// SIMATIC S7-200 project (STEP 7-Micro/WIN), CPU 226 CN REL 02.01

ORGANIZATION_BLOCK 主程序:OB1
TITLE=程序注释
BEGIN
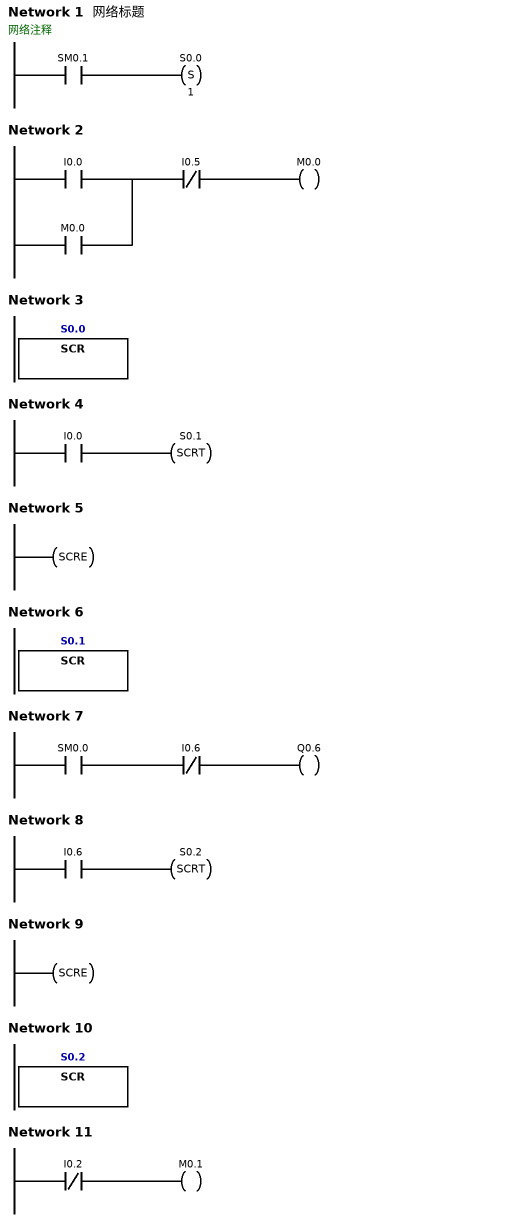
Network 1 // 网络标题
// 网络注释
LD     SM0.1
S      S0.0, 1
Network 2
LD     I0.0
O      M0.0
AN     I0.5
=      M0.0
Network 3
LSCR   S0.0
Network 4
LD     I0.0
SCRT   S0.1
Network 5
SCRE
Network 6
LSCR   S0.1
Network 7
LD     SM0.0
AN     I0.6
=      Q0.6
Network 8
LD     I0.6
SCRT   S0.2
Network 9
SCRE
Network 10
LSCR   S0.2
Network 11
LDN    I0.2
=      M0.1
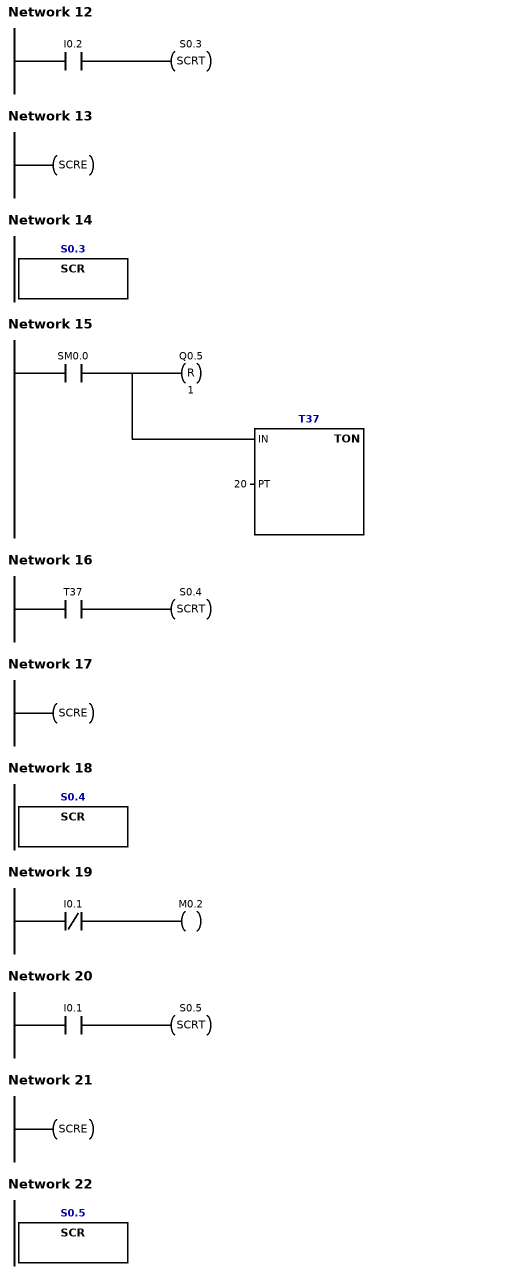
Network 12
LD     I0.2
SCRT   S0.3
Network 13
SCRE
Network 14
LSCR   S0.3
Network 15
LD     SM0.0
R      Q0.5, 1
TON    T37, 20
Network 16
LD     T37
SCRT   S0.4
Network 17
SCRE
Network 18
LSCR   S0.4
Network 19
LDN    I0.1
=      M0.2
Network 20
LD     I0.1
SCRT   S0.5
Network 21
SCRE
Network 22
LSCR   S0.5
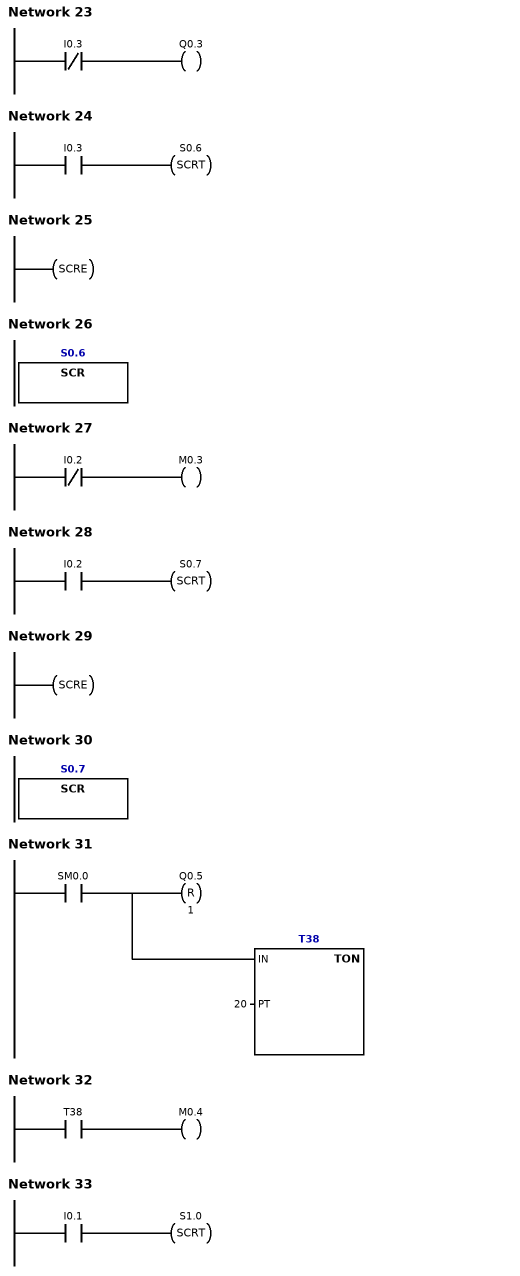
Network 23
LDN    I0.3
=      Q0.3
Network 24
LD     I0.3
SCRT   S0.6
Network 25
SCRE
Network 26
LSCR   S0.6
Network 27
LDN    I0.2
=      M0.3
Network 28
LD     I0.2
SCRT   S0.7
Network 29
SCRE
Network 30
LSCR   S0.7
Network 31
LD     SM0.0
R      Q0.5, 1
TON    T38, 20
Network 32
LD     T38
=      M0.4
Network 33
LD     I0.1
SCRT   S1.0
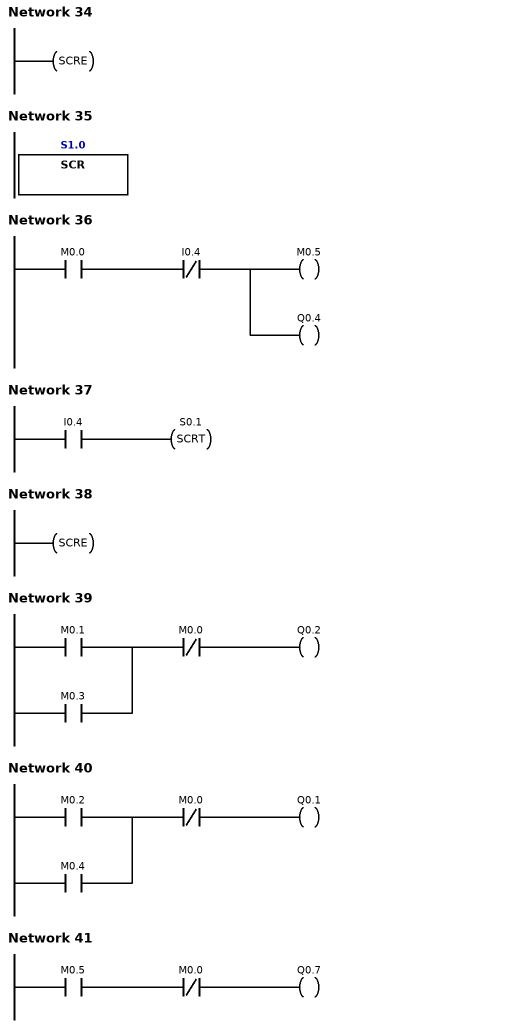
Network 34
SCRE
Network 35
LSCR   S1.0
Network 36
LD     M0.0
AN     I0.4
=      M0.5
=      Q0.4
Network 37
LD     I0.4
SCRT   S0.1
Network 38
SCRE
Network 39
LD     M0.1
O      M0.3
AN     M0.0
=      Q0.2
Network 40
LD     M0.2
O      M0.4
AN     M0.0
=      Q0.1
Network 41
LD     M0.5
AN     M0.0
=      Q0.7
END_ORGANIZATION_BLOCK
